# EPICS autosave request: iocBoot/ioc13bmd_DAC_XPS/auto_positions.req
file "CARS_motor_positions.req",         P=$(P), M=m89
file "CARS_motor_positions.req",         P=$(P), M=m90
file "CARS_motor_positions.req",         P=$(P), M=m91
